Fanuc KAREL source: kt00441.KL

PROGRAM KT00441
%NOLOCKGROUP
VAR
R1:REAL;I2:INTEGER;OUT:BOOLEAN
BEGIN
--
--
R1=2.0
I2=3
OUT=(R1>=I2)
END KT00441
